// Gets the lower bound index of the array of specified type.
FUNCTION F_GetDIntArrayLowerBound : T_Position // The lower bound index of the specified array.
VAR_IN_OUT
	arArray : ARRAY[*] OF DINT; // The array to query.
END_VAR

F_GetDIntArrayLowerBound := LOWER_BOUND(arArray, 1);

END_FUNCTION

(* stored: Version 1.1.0.1
   POU F_GetDIntArrayLowerBound: Id {198549b2-bba7-08a4-0f23-be66c10093d6}, SpecialFunc None *)
